// TIA Portal V20 export
VAR_GLOBAL   // PLC tag table "LER_E5CC"
END_VAR
VAR_GLOBAL CONSTANT   // user constants
   Number_Of_E5CC : Int := 5;
   E5CC_Lengths : Int := 20;
END_VAR
